// TIA Portal V18 export
VAR_GLOBAL   // PLC tag table "Default tag table"
   outtt AT %M0.0 : Bool;
END_VAR
